# EPICS substitutions: pvNotepadApp/Db/array_1.substitutions
#Substitution file for single record
file waveform.template
{
    pattern { RECORD                ,NELM}
            { $(HUTCH):NOTE:$(IDENTIFIER):ARRAY:01,$(NELM)}
}
